FUNCTION_BLOCK PUBLIC FB_STRINGS
VAR_INPUT
END_VAR
VAR_OUTPUT
END_VAR
VAR
END_VAR

METHOD PUBLIC IsNumeric : BOOL
VAR_INPUT
	In : STRING;
END_VAR
VAR
	i : USINT;
	NewString : STRING;
	Pos : INT;
END_VAR
IF In = '' THEN
	IsNumeric := FALSE;
ELSE
	NewString := In;
	IF FIND(NewString, '-') = 1 THEN
		NewString := DELETE(NewString, 1, 1);
	END_IF;
	FOR i := 0 TO 9 DO
		WHILE TRUE DO
			Pos := FIND(NewString, TO_STRING(i));
			IF Pos <> 0 THEN
				NewString := DELETE(NewString, 1, Pos);
			ELSE
				EXIT;
			END_IF;
		END_WHILE;
	END_FOR;
	IsNumeric := LEN(NewString) = 0;
END_IF
END_METHOD

END_FUNCTION_BLOCK

(* stored: Version 1.1.0.1, ProductVersion 3.1.4024.12
   POU FB_STRINGS: Id {96996496-049c-44ad-ad7b-599677ac70c2}, SpecialFunc None
   Method IsNumeric: Id {fbebf66f-840b-4244-9a2a-4b8885fa7770} *)
